FUNCTION MqttClient : FB_IotMqtt5Client
PROGRAM PrgMqttCom
VAR
    fbMqttClient    : FB_IotMqttClient;
    bSetParameter   : BOOL := TRUE;
    bConnect        : BOOL := TRUE;
END_VAR

// NETWORK 1

END_FUNCTION

(* stored: Version 1.1.0.1, ProductVersion 3.1.4024.12
   POU MqttClient: Id {adbe478c-a52c-44ac-8e07-ffa9326a6190}, SpecialFunc None *)
